(* CoDeSys 2.3.9.47 project: AdsMqtt.pro *)
(* Libraries: STANDARD.LIB 5.6.98 12:03:02 *)

(* Task configuration *)
TASK Standard (PRIORITY := 0, INTERVAL := T#10ms);
	MAIN
END_TASK

(* POU MAIN, ST *)
PROGRAM MAIN
VAR
   boolVal	: BOOL;
    intVal	: INT;
    dintVal	: DINT;
    sintVal	: SINT;
    lrealVal	: LREAL;
    realVal	: REAL;
    stringVal : STRING(10);
	i: INT;
END_VAR
i := i + 1;

IF boolval THEN
IF (i MOD 10 = 0) THEN
intVal := intVal + 1;
END_IF
ELSE
intVal := 0;
END_IF
END_PROGRAM
